TYPE DUT_SENSOR_DATAS_h8 :
UNION
	data_lreal:REAL;
	data_byte:ARRAY[0..3] OF BYTE;
END_UNION
END_TYPE

(* stored: Version 1.1.0.1, ProductVersion 3.1.4024.6
   DUT DUT_SENSOR_DATAS_h8: Id {1a31dcbf-9d5d-4f47-9fe4-6ec4411eb873} *)
